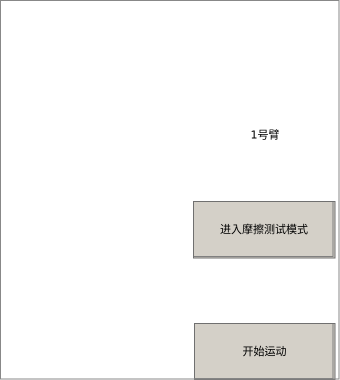
VISUALIZATION friction_a1  // 340x380
    Button (193,201 142x57), "进入摩擦测试模式", colour toggle: g_frictionTest.m_testMode[1]
        toggle g_frictionTest.m_testMode[1]
    Button (194,323 141x57), "开始运动", colour toggle: g_frictionTest.m_startMotion[1]
        toggle g_frictionTest.m_startMotion[1]
    Label (190,120 150x30), "1号臂"
END_VISUALIZATION

(* stored: Version 1.1.0.1, ProductVersion 3.1.4024.11
   Visu friction_a1: Id {5a775795-2dfc-41c7-a1ee-72e1b8a53633} *)
